(* PLC project Unnamed, Unknown Unnamed 1 *)
(* stored: creationDateTime 2026-09-20T16:11:10, modificationDateTime 2026-09-20T17:20:27 *)

PROGRAM TankFill
  VAR
    TankFillAuto_Cmd : BOOL;  (* Automatic fill latch/command *)
    TankValveOpen : BOOL;  (* Fill valve open command *)
    Estop_Cmd : BOOL;  (* Emergency-stop input *)
    TankLevelHi_Alarm : BOOL;  (* High-level alarm *)
    TankLevelLo_Alarm : BOOL;  (* Low-level alarm *)
    TankLevel_LIT : REAL := 5.0;  (* Tank level in feet *)
    TankEmpty_SP : REAL := 2.0;  (* Fill start setpoint *)
    TankFull_SP : REAL := 8.0;  (* Fill stop setpoint *)
    TankLoAlarm_SP : REAL := 1.0;  (* Low alarm setpoint *)
    TankHiAlarm_SP : REAL := 9.0;  (* High alarm setpoint *)
  END_VAR

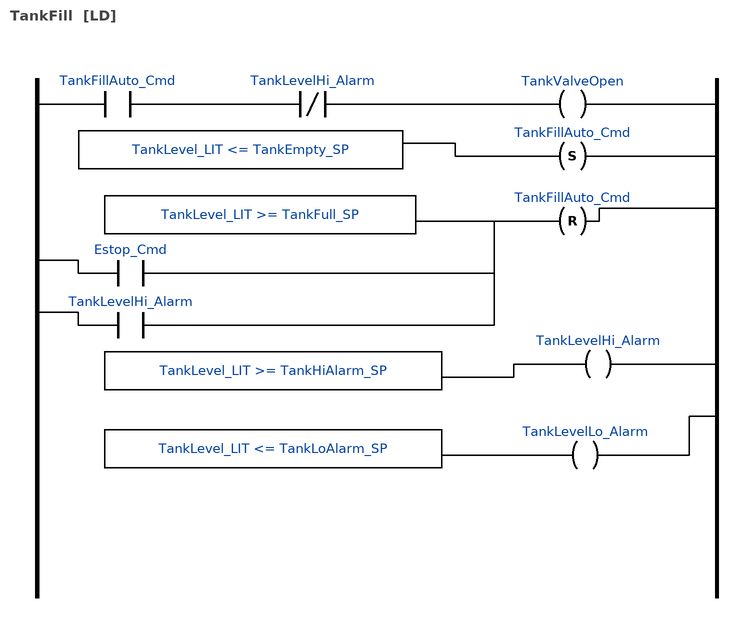
(* LD diagram, written out as Structured Text *)
TankValveOpen := TankFillAuto_Cmd AND NOT TankLevelHi_Alarm;
IF TankLevel_LIT <= TankEmpty_SP THEN TankFillAuto_Cmd := TRUE; END_IF;
IF Estop_Cmd OR (TankLevel_LIT >= TankFull_SP) OR TankLevelHi_Alarm THEN TankFillAuto_Cmd := FALSE; END_IF;
TankLevelHi_Alarm := TankLevel_LIT >= TankHiAlarm_SP;
TankLevelLo_Alarm := TankLevel_LIT <= TankLoAlarm_SP;
END_PROGRAM

CONFIGURATION Config0
  RESOURCE Res0 ON PLC
    TASK task0(INTERVAL := T#20ms, PRIORITY := 0);
    PROGRAM instance0 WITH task0 : TankFill;
  END_RESOURCE
END_CONFIGURATION
